(* CoDeSys 2.3 export: STRPLC160AI.EXP *)

(* Data type *)
TYPE strPLC160AI :
(*
	поз. А1
	Контроллер ПЛК160
	Аналоговые входы
*)
STRUCT
	UZSignal : ARRAY [1..MAX_UZ_NUM] OF tUZSignal;
(*
	Аналоговые входы №1-3:
	Сигналы 0-20mA от частотных преобразователей UZ
*)

	DilutionSignal : ARRAY [1..MAX_BOILERS_NUM] OF tDelutionSignal;
(*
	Аналоговые входы №4-6:
	Сигналы 4-20mA измерения разрежения из щита ЩИР
	по одному сигналу на каждый котел
*)

	Reserved : ARRAY [1..2] OF tAnalogInput;
(*
	Незадействованные входы
*)


END_STRUCT
END_TYPE
